FUNCTION Runtime

IF _Runtime.iFirstCyclic <> 0 THEN
	_Runtime.iFirstCyclic.Exe();
END_IF

END_FUNCTION

(* stored: Version 1.1.0.1
   POU Runtime: Id {8fe3d9a9-21d6-4789-9d5e-2d045d4180e3}, SpecialFunc None *)
